Staubli VAL3: msgBoxDisplay.pgx

public program msgBoxDisplay(num x_nBoxWidth)
  local num l_i
  local string l_sLine
  local string l_sEmptyLine
  local string l_sGraphicLine
begin
  // This program displays a message box on the MCP
  //
  // Input param
  // nTxtBoxRow      : Message to display
  // nTxtBoxCol      : width of the message box to display
  //
  // Output param
  //
  // Created 23-02-05                           C.CURRIVAND
  //------------------------------------------------------------------
  //
  l_sEmptyLine="                                        "
  l_sGraphicLine="────────────────────────────────────────"
  //
  // display upper graphic line
  l_sLine="┌"+mid(l_sGraphicLine,x_nBoxWidth-2,1)+"┐"
  call type(nTxtBoxCol,nTxtBoxRow,l_sLine)
  //
  //display message
  for l_i=0 to size(sWrkString)-1
    if (x_nBoxWidth-len(sWrkString[l_i])>=0)
      l_sLine="│"+sWrkString[l_i]+mid(l_sEmptyLine,x_nBoxWidth-2-len(sWrkString[l_i]),1)+"│"
    else
      l_sLine="│"+sWrkString[l_i]+"│"
    endIf
    call type(nTxtBoxCol,nTxtBoxRow+1+l_i,l_sLine)
  endFor
  // display lower graphic line
  l_sLine="└"+mid(l_sGraphicLine,x_nBoxWidth-2,1)+"┘"
  call type(nTxtBoxCol,nTxtBoxRow+1+l_i,l_sLine)
  //
end
